FUNCTION_BLOCK FB_AC_Mitsubishi EXTENDS FB_AirConditionerBase
VAR_INPUT
END_VAR
VAR_OUTPUT
END_VAR
VAR
END_VAR

METHOD HandleMessage : BOOL
VAR_INPUT
	message :STRING;
END_VAR
IF message='turnedOff' THEN
	ADSLOGSTR(msgCtrlMask := ADSLOG_MSGTYPE_ERROR, msgFmtStr := 'Mitsubishi Air Conditioner Turned Off', strArg := '');
END_IF
END_METHOD

END_FUNCTION_BLOCK

(* stored: Version 1.1.0.1, ProductVersion 3.1.4024.9
   POU FB_AC_Mitsubishi: Id {a48e41b7-d9d4-41f3-b36e-7cc65cd7c5f3}, SpecialFunc None
   Method HandleMessage: Id {b55e9228-c000-463b-b230-3ca225c0cf46} *)
